INTERFACE ITask

METHOD Abort : BOOL
VAR_INPUT
END_VAR
END_METHOD

PROPERTY Busy : bool
GET
END_GET
END_PROPERTY

PROPERTY Done : bool
GET
END_GET
END_PROPERTY

PROPERTY Error : bool
GET
END_GET
END_PROPERTY

END_INTERFACE

(* stored: Version 1.1.0.1, ProductVersion 3.1.4024.12
   Itf ITask: Id {c30402e0-3599-4862-bb6b-454152446820}
   Method Abort: Id {80de65a5-defe-42ef-8f5d-8143dafab5d7}
   Property Busy: Id {d320d1fd-45b2-4aad-ad9b-94759823337c}
   Get Get: Id {8ea5b166-32f2-412b-b338-ee8edca7ef40}
   Property Done: Id {9d22b659-8f04-42b3-8f6b-1e7f626a9631}
   Get Get: Id {0f443cdb-2eef-4138-b1c9-b0ce7512d455}
   Property Error: Id {1aa21dfd-89ca-448a-9552-890b89b0aabf}
   Get Get: Id {c5a78472-4a69-4cc5-bad2-f6a03405ae35} *)
